Staubli VAL3: changeSession.pgx

public program changeSession(string x_sName)
  local string l_sPathTraj
  local string l_sPathProg
  local string l_sRootPath
  local string l_sPathCycle
  local string l_sPathSave
  local num i
begin
  //
  // change the session
  //
  // check if the robot is empty
  if (isEmpty()and isSettled())and watch(bToReload==false,120)==true
    if x_sName!="template"
      l_sPathTraj="saveTraj/"
      l_sPathProg="saveProg/"
      l_sPathSave="saveCycle/"
      l_sRootPath="Disk://session/"+x_sName+"/"
      // trajectory
      sPathTraj=l_sRootPath+l_sPathTraj
      // program
      sPathProg=l_sRootPath+l_sPathProg
      // process list
      sPathPList=l_sRootPath+l_sPathSave
      // save it
      sSession=x_sName
    else
      // trajectory
      sPathTraj="kernel/template/session/saveTraj/"
      // program
      sPathProg="kernel/template/session/saveProg/"
      // process list
      sPathPList="kernel/template/session/saveCycle/"
    endIf
    // reaload all...
    bToReload=true
    // watch it
    if watch(bToReload==false,120)==false
      popUpMsg("ERROR TIMEOUT!!! LOADING SESSION ...")
      logMsg("ERROR LOADING SESSION ...")
      wait(bToReload==false)
    endIf
  else
    popUpMsg("Error while changing the session the robot is working...")
    logMsg("Error while changing the session the robot is working...")
    delay(1)
  endIf
end
